FUNCTION_BLOCK TUnitTestUnderTest EXTENDS TUnitTestBase
VAR_INPUT
END_VAR
VAR_OUTPUT
END_VAR
VAR
END_VAR

END_FUNCTION_BLOCK

(* stored: Version 1.1.0.1, ProductVersion 3.1.4024.4
   POU TUnitTestUnderTest: Id {cb7c53df-47d6-4f3a-8c1a-bbc9f9ec13cf}, SpecialFunc None *)
